FUNCTION_BLOCK "__jxd1_home"
TITLE = {"status":"current","deprecatedBy": null,"dependencies":["jxd1_driveUnit_16bytes_directNumericalSettingModePdi","jxd1_driveUnit_16bytes_directNumericalSettingModePdo","TON_TIME"]}
{ S7_Optimized_Access := 'TRUE' }
AUTHOR : cyanezf
FAMILY : 'core/controller/smc/jxd1'
NAME : __jxd1_home
VERSION : 1.0

   VAR_INPUT
      request { ExternalWritable := 'False'} : Bool;   // IR: 1=Request
      abort { ExternalWritable := 'False'} : Bool;   // IR: 1=Abort positioning
      ready { ExternalAccessible := 'False'; ExternalVisible := 'False'; ExternalWritable := 'False'} : Bool;   // IX: 1=Ready
   END_VAR
   VAR_INPUT RETAIN
      watchdogTime : Time := T#1M;   // IW: Watchdog time
      isHomedByCalcTime : Time := T#100ms;   // IW: Time to delay Is homed by calculation
      homePosition : LReal;   // IW: Home position
      homeTolerance : LReal := 1.0;   // IW: Home tolerance
   END_VAR

   VAR_OUTPUT
      status { ExternalWritable := 'False'} : Int;   // OR: Status code. See constants
      busy { ExternalWritable := 'False'} : Bool;   // OR: 1=Busy (some action)
      done { ExternalWritable := 'False'} : Bool;   // OR: 1=Done
      error { ExternalWritable := 'False'} : Bool;   // OR: 1=Error
      commandAborted { ExternalWritable := 'False'} : Bool;   // OR: 1=Command aborted
   END_VAR

   VAR_IN_OUT
      actualPosition { ExternalAccessible := 'False'; ExternalVisible := 'False'; ExternalWritable := 'False'} : LReal;   // IOX: Read only - Actual position
      pdi : "jxd1_driveUnit_16bytes_directNumericalSettingModePdi";   // IOX: Read only - PDI
      pdo : "jxd1_driveUnit_16bytes_directNumericalSettingModePdo";   // IOX: Conditional Partial Write - PDO
   END_VAR

   VAR
      step { ExternalWritable := 'False'} : Int := #STEP_0_IDLE;   // SR: Step
      private { ExternalAccessible := 'False'; ExternalVisible := 'False'; ExternalWritable := 'False'} : Struct   // SX: Private static variables
         request { ExternalAccessible := 'False'; ExternalVisible := 'False'; ExternalWritable := 'False'} : Bool;
         isHomedByPdi { ExternalAccessible := 'False'; ExternalVisible := 'False'; ExternalWritable := 'False'} : Bool;
         watchdogTimer {InstructionName := 'TON_TIME'; LibVersion := '1.0'; ExternalAccessible := 'False'; ExternalVisible := 'False'; ExternalWritable := 'False'; S7_SetPoint := 'False'} : TON_TIME;
         isHomedByCalcTimer {InstructionName := 'TON_TIME'; LibVersion := '1.0'; ExternalAccessible := 'False'; ExternalVisible := 'False'; ExternalWritable := 'False'; S7_SetPoint := 'False'} : TON_TIME;
      END_STRUCT;
   END_VAR

   VAR_TEMP
      aux : Bool;
      isHomedByPdiPulse : Bool;
      isHomedByCalc : Bool;
      requestPulseOn : Bool;
   END_VAR

   VAR CONSTANT
      STATUS_0000_IDLE : Int := 0;
      STATUS_0001_DONE : Int := 1;
      STATUS_6000_BUSY : Int := 16#6000;
      STATUS_8000_ABORTED : Int := 16#8000;
      STATUS_8001_DRIVE_ERROR : Int := 16#8001;
      STEP_0_IDLE : Int := 0;
      STEP_1_REQ : Int := 1;
      STEP_2_BUSY : Int := 2;
      STEP_3_DONE : Int := 3;
      STEP_20_ABORTED : Int := 20;
      STEP_21_ERROR : Int := 21;
   END_VAR


BEGIN
(*--
# Documentation

## Log

| version | date | author | description |
|:-------:|:----:|:------:|:------------|
| v1.0 | 2026-07-19 | cyanezf | First version |

## Description

This private function block implements the home logic for the SMC JXD1 step motor controller. It provides a controlled way to home the motor, ensuring that it reaches the home position within the specified tolerance. The function block uses a state machine to manage the homing process, including holding the motor for a specified time before turning off the servo.

--*)

	// Request Event
	#requestPulseOn := #request AND NOT #private.request;
	#private.request := #request;

	// Is homed by PDI
	#isHomedByPdiPulse := #pdi.status.isHomed AND NOT #private.isHomedByPdi;
	#private.isHomedByPdi := #pdi.status.isHomed;

	// Is homed by calculation
	#aux :=#pdi.status.isHomed AND ABS(#actualPosition - #homePosition) <= #homeTolerance  AND #step = #STEP_2_BUSY;
	#private.isHomedByCalcTimer(IN:=#aux,
	PT:=#isHomedByCalcTime,
	Q=>#isHomedByCalc);

	REGION Unconditional transitions

	  // ############################################################################
	  IF NOT #ready THEN
	    IF #step >= #STEP_1_REQ AND #step <= #STEP_2_BUSY THEN
	      #step := #STEP_21_ERROR;
	    END_IF;

	    // ############################################################################
	  ELSIF #abort THEN
	    IF #step >= #STEP_1_REQ AND #step <= #STEP_2_BUSY THEN
	      #step := #STEP_20_ABORTED;
	    END_IF;

	  END_IF;

	END_REGION

	REGION Steps

	  IF #step = #STEP_0_IDLE THEN

	    // Status
	    #status := #STATUS_0000_IDLE;
	    #busy := 0;
	    #done := 0;
	    #error := 0;
	    #commandAborted := 0;

	    IF #request AND #ready AND NOT #pdi.status.isRunning THEN
	      #step := #STEP_1_REQ;
	    END_IF;
	  END_IF;

	  // ############################################################################
	  // Normal task steps
	  // ############################################################################
	  IF #step = #STEP_1_REQ THEN

	    // Status
	    #status := #STATUS_6000_BUSY;
	    #busy := 1;
	    #done := 0;
	    #error := 0;
	    #commandAborted := 0;

	    // Init flags
	    // Homing
	    #pdo.control.homing := 1;
	    // Jog
	    #pdo.control.jogMinus := 0;
	    #pdo.control.jogPlus := 0;
	    #pdo.control.flight := 0;
	    // Push
	    #pdo.control.push := 0;
	    #pdo.control.pushDirection := 0;
	    // Abs
	    #pdo.control.incMode := 0;
	    // Start abs
	    #pdo.control.start := 0;

	    // Transitions
	    IF #pdi.status.isRunning THEN
	      #step := #STEP_2_BUSY;
	    END_IF;

	    // ############################################################################
	  ELSIF #step = #STEP_2_BUSY THEN

	    // Update
	    #pdo.control.homing := 0;

	    // Transitions
	    IF #isHomedByPdiPulse OR #isHomedByCalc THEN
	      #step := #STEP_3_DONE;
	    END_IF;

	    // ############################################################################
	  ELSIF #step = #STEP_3_DONE THEN

	    // Status
	    #status := #STATUS_0001_DONE;
	    #busy := 0;
	    #done := 1;
	    #error := 0;
	    #commandAborted := 0;

	    // Transitions
	    IF NOT #request THEN
	      #step := #STEP_0_IDLE;
	    END_IF;

	  END_IF;

	  // ############################################################################
	  // Abort and error steps
	  // ############################################################################
	  IF #step = #STEP_20_ABORTED THEN

	    // Status
	    #status := #STATUS_8000_ABORTED;
	    #busy := 0;
	    #done := 0;
	    #error := 0;
	    #commandAborted := 1;

	    // Transitions
	    IF NOT #abort THEN
	      #step := #STEP_0_IDLE;
	    END_IF;

	    // ############################################################################
	  ELSIF #step = #STEP_21_ERROR THEN

	    // Status
	    #status := #STATUS_8001_DRIVE_ERROR;
	    #busy := 0;
	    #done := 0;
	    #error := 1;
	    #commandAborted := 0;

	    // Transitions
	    IF NOT #request THEN
	      #step := #STEP_0_IDLE;
	    END_IF;

	  END_IF;

	END_REGION

	ENO := true;

END_FUNCTION_BLOCK

